{attribute addProperty BoxType "AX8118-0000-0041-0041"}
{attribute addProperty Id "DeviceDevice_FD48B4B01620Ch_ACh_A_99F8614F240300WcStateAT %I*WcState_F855686C1620InfoDataAT %I*InfoData_F030DC9B200250"}
{attribute addProperty CRC "218904718"}
{attribute addProperty SizeInBites "472"}
{attribute addProperty SizeInBytes "59"}
TYPE AX8118_A2FEB36A :
STRUCT
	{attribute addProperty Name "Device"}
	Device : Device_FD48B4B0;
	{attribute addProperty Name "Ch_A"}
	Ch_A : Ch_A_99F8614F;
	{attribute addProperty Name "WcState"}
	WcState : WcState_F855686C;
	{attribute addProperty Name "InfoData"}
	InfoData : InfoData_F030DC9B;
END_STRUCT
END_TYPE

(* stored: Version 1.2.0.0, ProductVersion 3.1.4024.9
   DUT AX8118_A2FEB36A: Id {2f25dcd9-da57-4d4b-8487-56b04fcc37d5} *)
